TYPE ST_Results : 
STRUCT
END_STRUCT
END_TYPE

(* stored: DUT ST_Results: Id a28eba75-c787-4fd2-bac5-d2b34f4a1fc4 *)
